{attribute addProperty BoxType "KL1212"}
{attribute addProperty Id "InputAT %I*BOOL000ErrorAT %I*BOOL000PowerAT %Q*BOOL000"}
{attribute addProperty CRC "3705944467"}
{attribute addProperty SizeInBites "0"}
{attribute addProperty SizeInBytes "0"}
TYPE Channel_DCE43993 :
STRUCT
	{attribute addProperty Name "Input"}
	Input AT %I* : BOOL;
	{attribute addProperty Name "Error"}
	Error AT %I* : BOOL;
	{attribute addProperty Name "Power"}
	Power AT %Q* : BOOL;
END_STRUCT
END_TYPE

(* stored: Version 1.2.0.0, ProductVersion 3.1.4024.9
   DUT Channel_DCE43993: Id {b89b214b-545f-478c-b5e9-03dc7364ef53} *)
